// Mitsubishi GX Works2 project: DATN   PLC: FX3U/FX3UC

PROGRAM MAIN
VAR
  Retrieval_1 : Retrieval;
  Storage : Storage;
  Home_Sto_1 : Home_Sto;
  GoToFailPos_1 : GoToFailPos;
END_VAR
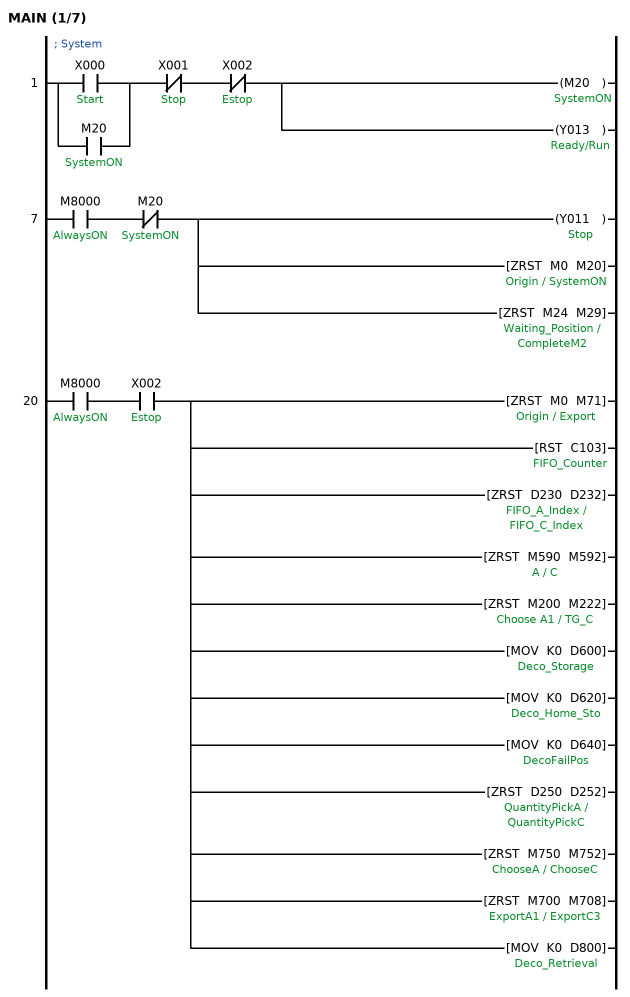
; System
1     LD      X000  ; Start
      OR      M20  ; SystemON
      ANI     X001  ; Stop
      ANI     X002  ; Estop
      OUT     M20  ; SystemON
      OUT     Y013  ; Ready/Run
7     LD      M8000  ; AlwaysON
      ANI     M20  ; SystemON
      OUT     Y011  ; Stop
      ZRST    M0 M20  ; Origin
      ZRST    M24 M29  ; Waiting_Position / CompleteM2
20    LD      M8000  ; AlwaysON
      AND     X002  ; Estop
      ZRST    M0 M71  ; Export
      RST     C103  ; FIFO_Counter
      ZRST    D230 D232  ; FIFO_A_Index / FIFO_C_Index
      ZRST    M590 M592  ; A / C
      ZRST    M200 M222  ; Choose A1 / TG_C
      MOV     K0 D600  ; Deco_Storage
      MOV     K0 D620  ; Deco_Home_Sto
      MOV     K0 D640  ; DecoFailPos
      ZRST    D250 D252  ; QuantityPickA / QuantityPickC
      ZRST    M750 M752  ; ChooseA / ChooseC
      ZRST    M700 M708  ; ExportA1 / ExportC3
      MOV     K0 D800  ; Deco_Retrieval
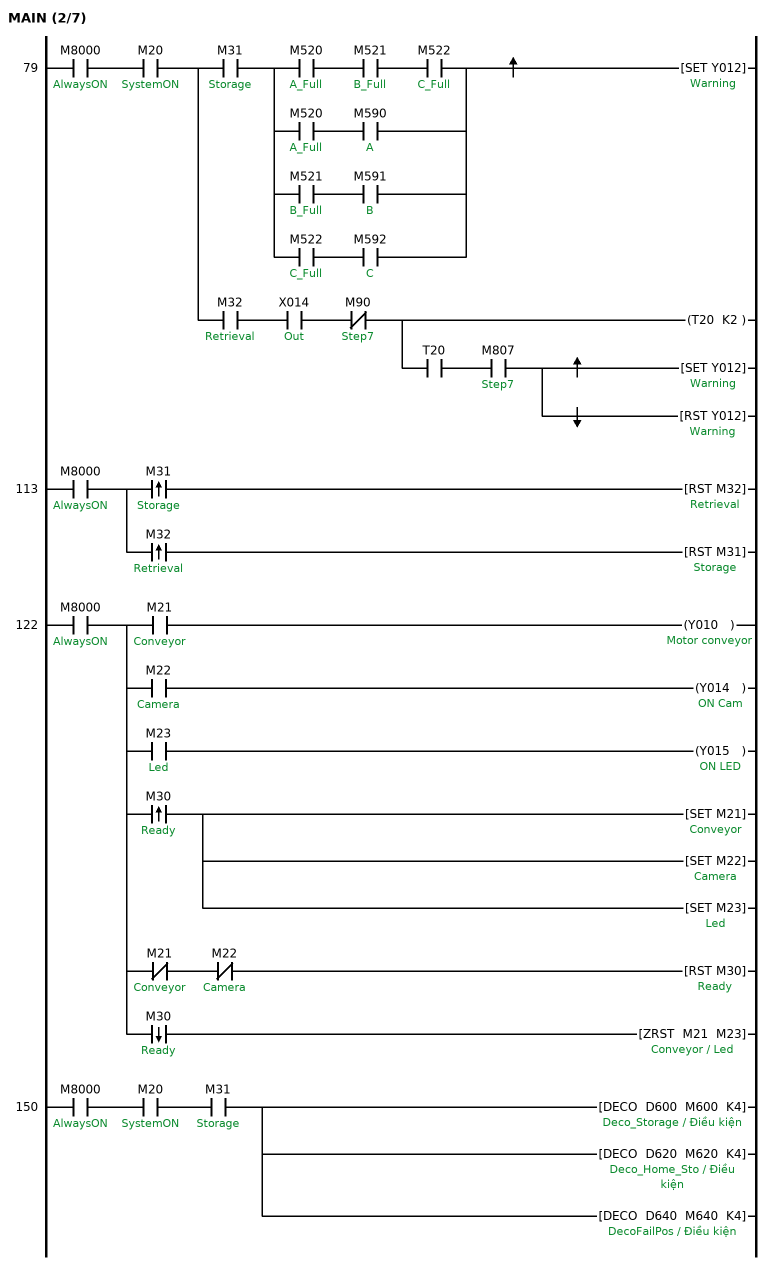
79    LD      M8000  ; AlwaysON
      AND     M20  ; SystemON
      MPS
      AND     M31  ; Storage
      LD      M520  ; A_Full
      AND     M521  ; B_Full
      AND     M522  ; C_Full
      LD      M520  ; A_Full
      AND     M590  ; A
      ORB
      LD      M521  ; B_Full
      AND     M591  ; B
      ORB
      LD      M522  ; C_Full
      AND     M592  ; C
      ORB
      ANB
      MEP
      SET     Y012  ; Warning
      MPP
      AND     M32  ; Retrieval
      AND     X014  ; Out
      ANI     M90  ; Step7
      OUT     T20 K2
      AND     T20
      AND     M807  ; Step7
      MPS
      MEP
      SET     Y012  ; Warning
      MPP
      MEF
      RST     Y012  ; Warning
113   LD      M8000  ; AlwaysON
      MPS
      ANDP    M31  ; Storage
      RST     M32  ; Retrieval
      MPP
      ANDP    M32  ; Retrieval
      RST     M31  ; Storage
122   LD      M8000  ; AlwaysON
      MPS
      AND     M21  ; Conveyor
      OUT     Y010  ; Motor conveyor
      MRD
      AND     M22  ; Camera
      OUT     Y014  ; ON Cam
      MRD
      AND     M23  ; Led
      OUT     Y015  ; ON LED
      MRD
      ANDP    M30  ; Ready
      SET     M21  ; Conveyor
      SET     M22  ; Camera
      SET     M23  ; Led
      MRD
      ANI     M21  ; Conveyor
      ANI     M22  ; Camera
      RST     M30  ; Ready
      MPP
      ANDF    M30  ; Ready
      ZRST    M21 M23
150   LD      M8000  ; AlwaysON
      AND     M20  ; SystemON
      AND     M31  ; Storage
      DECO    D600 M600 K4  ; Điều kiện
      DECO    D620 M620 K4  ; Điều kiện
      DECO    D640 M640 K4  ; Điều kiện
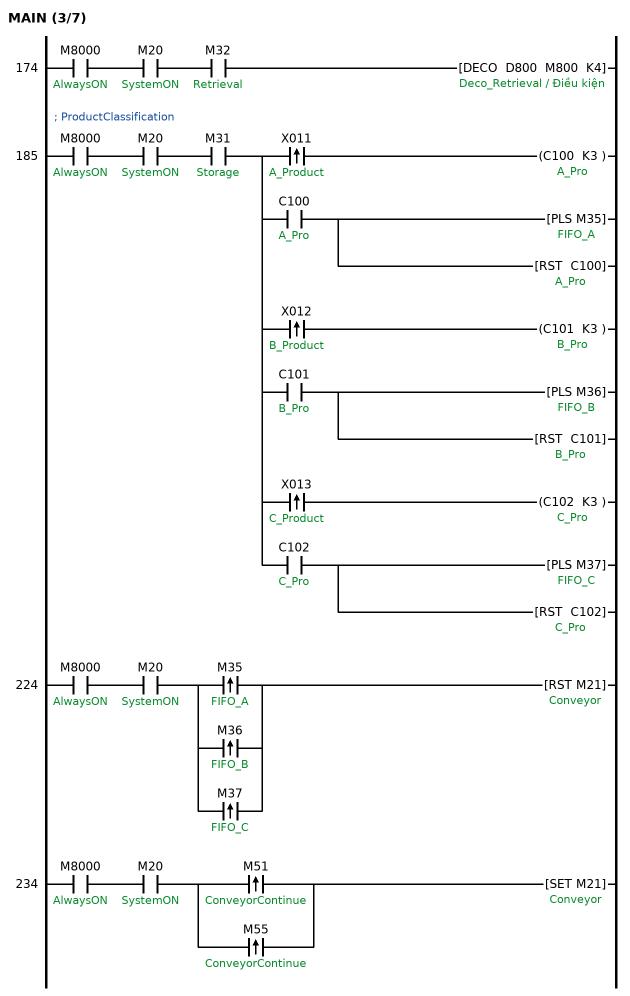
174   LD      M8000  ; AlwaysON
      AND     M20  ; SystemON
      AND     M32  ; Retrieval
      DECO    D800 M800 K4  ; Điều kiện
; ProductClassification
185   LD      M8000  ; AlwaysON
      AND     M20  ; SystemON
      AND     M31  ; Storage
      MPS
      ANDP    X011  ; A_Product
      OUT     C100 K3  ; A_Pro
      MRD
      AND     C100  ; A_Pro
      PLS     M35  ; FIFO_A
      RST     C100  ; A_Pro
      MRD
      ANDP    X012  ; B_Product
      OUT     C101 K3  ; B_Pro
      MRD
      AND     C101  ; B_Pro
      PLS     M36  ; FIFO_B
      RST     C101  ; B_Pro
      MRD
      ANDP    X013  ; C_Product
      OUT     C102 K3  ; C_Pro
      MPP
      AND     C102  ; C_Pro
      PLS     M37  ; FIFO_C
      RST     C102  ; C_Pro
224   LD      M8000  ; AlwaysON
      AND     M20  ; SystemON
      LDP     M35  ; FIFO_A
      ORP     M36  ; FIFO_B
      ORP     M37  ; FIFO_C
      ANB
      RST     M21  ; Conveyor
234   LD      M8000  ; AlwaysON
      AND     M20  ; SystemON
      LDP     M51  ; ConveyorContinue
      ORP     M55  ; ConveyorContinue
      ANB
      SET     M21  ; Conveyor
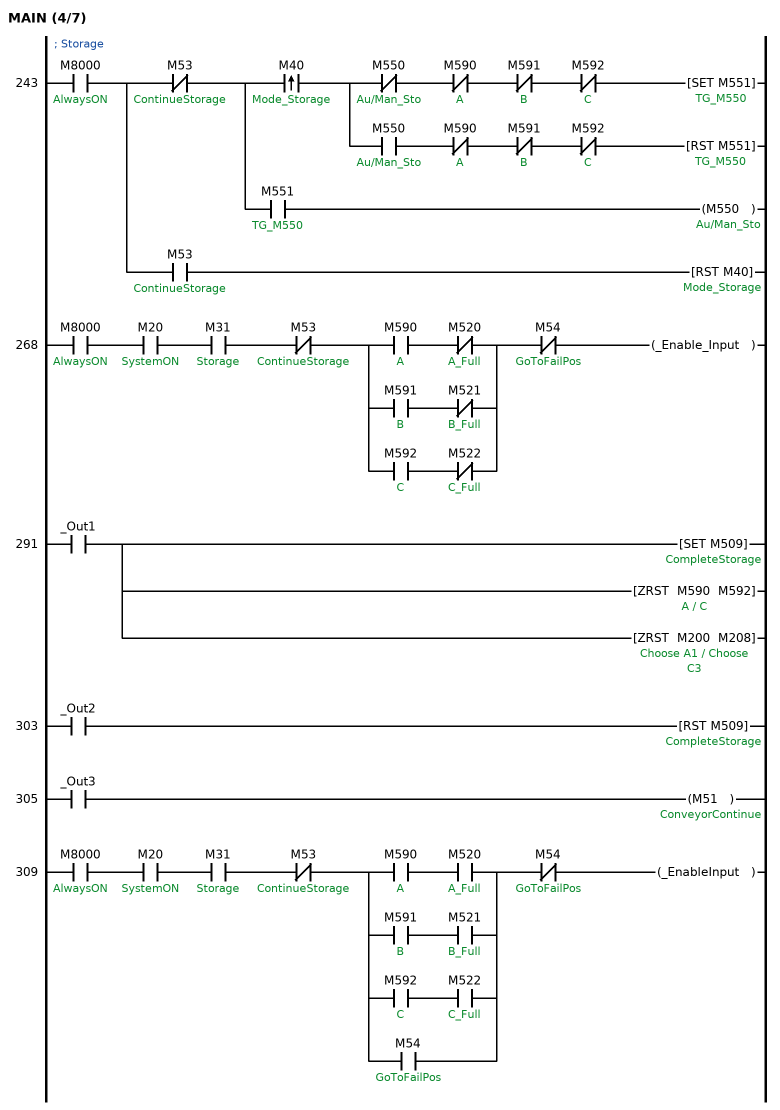
; Storage
243   LD      M8000  ; AlwaysON
      MPS
      ANI     M53  ; ContinueStorage
      MPS
      ANDP    M40  ; Mode_Storage
      MPS
      ANI     M550  ; Au/Man_Sto
      ANI     M590  ; A
      ANI     M591  ; B
      ANI     M592  ; C
      SET     M551  ; TG_M550
      MPP
      AND     M550  ; Au/Man_Sto
      ANI     M590  ; A
      ANI     M591  ; B
      ANI     M592  ; C
      RST     M551  ; TG_M550
      MPP
      AND     M551  ; TG_M550
      OUT     M550  ; Au/Man_Sto
      MPP
      AND     M53  ; ContinueStorage
      RST     M40  ; Mode_Storage
; FB BLK START Storage(Storage)
268   LD      M8000  ; AlwaysON
      AND     M20  ; SystemON
      AND     M31  ; Storage
      ANI     M53  ; ContinueStorage
      LD      M590  ; A
      ANI     M520  ; A_Full
      LD      M591  ; B
      ANI     M521  ; B_Full
      ORB
      LD      M592  ; C
      ANI     M522  ; C_Full
      ORB
      ANB
      ANI     M54  ; GoToFailPos
      OUT     _Enable_Input
; FB START
; FB_NAME Storage
; INSTANCE_NAME Storage
; FB IN_B:Enable_Input
; FB OUT_Out1:B
; FB OUT_Out2:B
; FB OUT_Out3:B
; FB END
291   LD      _Out1
      SET     M509  ; CompleteStorage
      ZRST    M590 M592
      ZRST    M200 M208  ; Choose C3
303   LD      _Out2
      RST     M509  ; CompleteStorage
305   LD      _Out3
      OUT     M51  ; ConveyorContinue
; FB BLK END
; FB BLK START Home_Sto(Home_Sto_1)
309   LD      M8000  ; AlwaysON
      AND     M20  ; SystemON
      AND     M31  ; Storage
      ANI     M53  ; ContinueStorage
      LD      M590  ; A
      AND     M520  ; A_Full
      LD      M591  ; B
      AND     M521  ; B_Full
      ORB
      LD      M592  ; C
      AND     M522  ; C_Full
      ORB
      OR      M54  ; GoToFailPos
      ANB
      ANI     M54  ; GoToFailPos
      OUT     _EnableInput
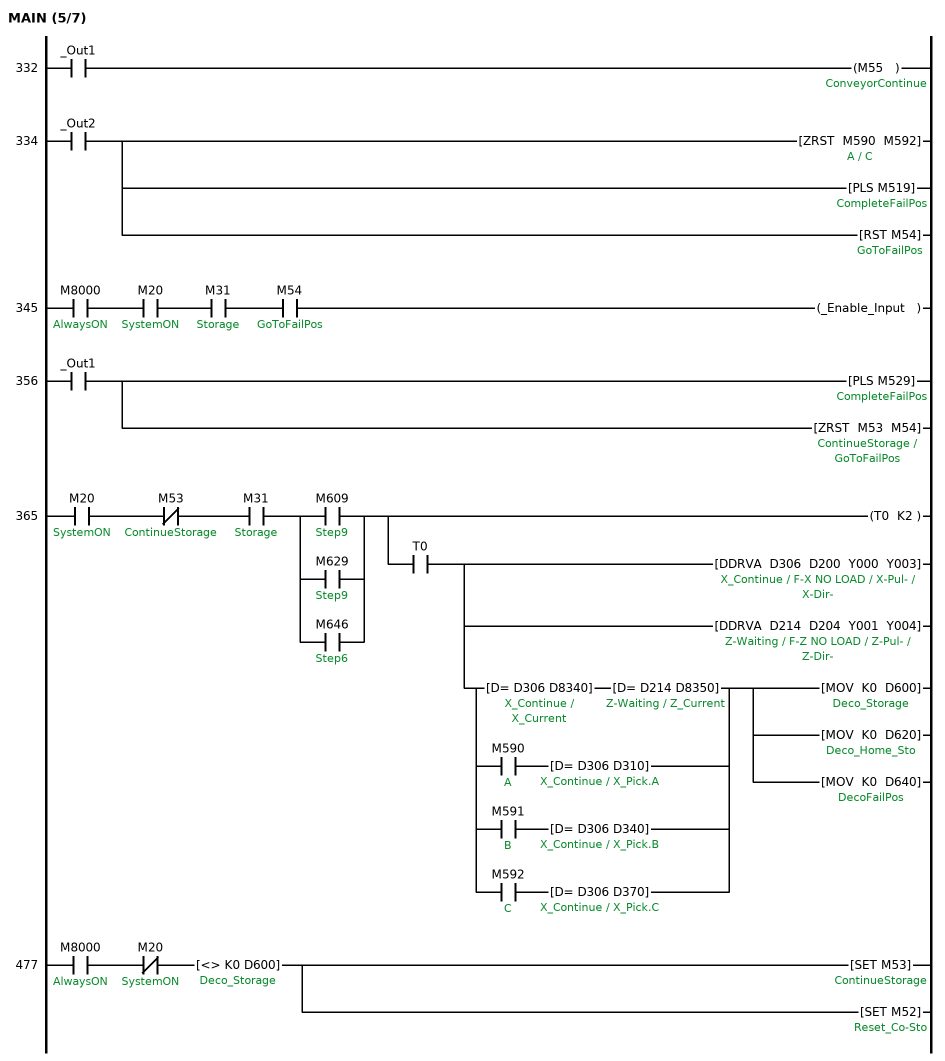
; FB START
; FB_NAME Home_Sto
; INSTANCE_NAME Home_Sto_1
; FB IN_B:EnableInput
; FB OUT_Out1:B
; FB OUT_Out2:B
; FB END
332   LD      _Out1
      OUT     M55  ; ConveyorContinue
334   LD      _Out2
      ZRST    M590 M592
      PLS     M519  ; CompleteFailPos
      RST     M54  ; GoToFailPos
; FB BLK END
; FB BLK START GoToFailPos(GoToFailPos_1)
345   LD      M8000  ; AlwaysON
      AND     M20  ; SystemON
      AND     M31  ; Storage
      AND     M54  ; GoToFailPos
      OUT     _Enable_Input
; FB START
; FB_NAME GoToFailPos
; INSTANCE_NAME GoToFailPos_1
; FB IN_B:Enable_Input
; FB OUT_Out1:B
; FB END
356   LD      _Out1
      PLS     M529  ; CompleteFailPos
      ZRST    M53 M54
; FB BLK END
365   LD      M20  ; SystemON
      ANI     M53  ; ContinueStorage
      AND     M31  ; Storage
      LD      M609  ; Step9
      OR      M629  ; Step9
      OR      M646  ; Step6
      ANB
      OUT     T0 K2
      AND     T0
      DDRVA   D306 D200 Y000 Y003  ; X_Continue / F-X NO LOAD / X-Pul- / X-Dir-
      DDRVA   D214 D204 Y001 Y004  ; Z-Waiting / F-Z NO LOAD / Z-Pul- / Z-Dir-
      LDD=    D306 D8340  ; X_Continue / X_Current
      ANDD=   D214 D8350  ; Z-Waiting / Z_Current
      LD      M590  ; A
      ANDD=   D306 D310  ; X_Continue / X_Pick.A
      ORB
      LD      M591  ; B
      ANDD=   D306 D340  ; X_Continue / X_Pick.B
      ORB
      LD      M592  ; C
      ANDD=   D306 D370  ; X_Continue / X_Pick.C
      ORB
      ANB
      MOV     K0 D600
      MOV     K0 D620
      MOV     K0 D640
477   LD      M8000  ; AlwaysON
      ANI     M20  ; SystemON
      AND<>   K0 D600  ; Deco_Storage
      SET     M53  ; ContinueStorage
      SET     M52  ; Reset_Co-Sto
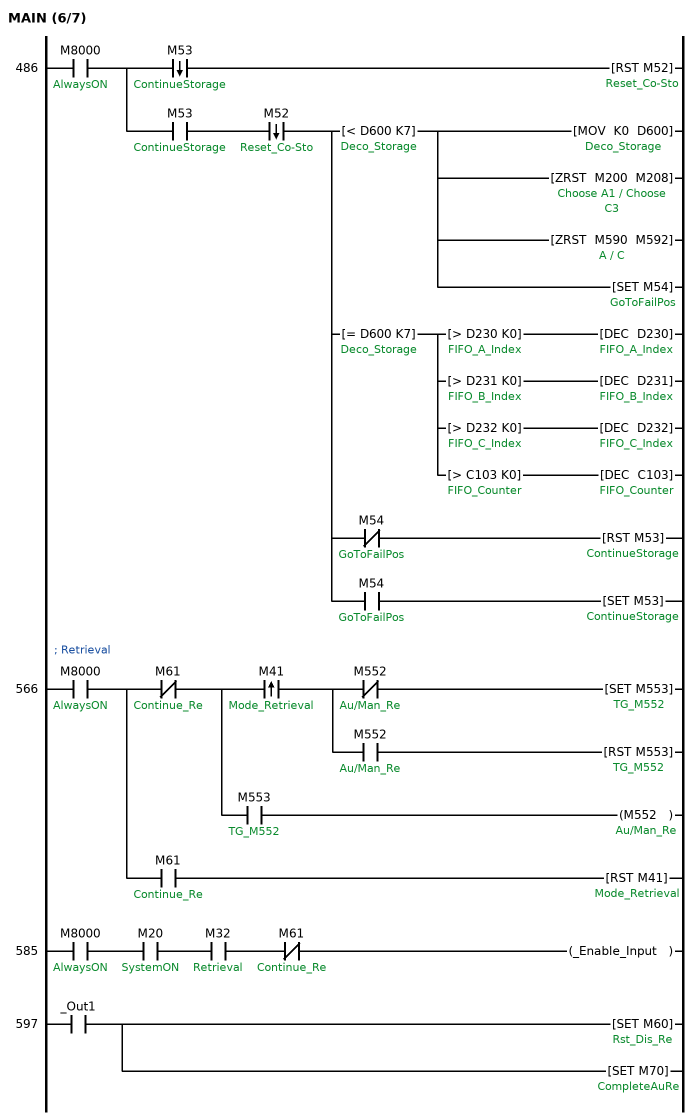
486   LD      M8000  ; AlwaysON
      MPS
      ANDF    M53  ; ContinueStorage
      RST     M52  ; Reset_Co-Sto
      MPP
      AND     M53  ; ContinueStorage
      ANDF    M52  ; Reset_Co-Sto
      MPS
      AND<    D600 K7  ; Deco_Storage
      MOV     K0 D600
      ZRST    M200 M208
      ZRST    M590 M592
      SET     M54  ; GoToFailPos
      MRD
      AND=    D600 K7  ; Deco_Storage
      MPS
      AND>    D230 K0  ; FIFO_A_Index
      DEC     D230
      MRD
      AND>    D231 K0  ; FIFO_B_Index
      DEC     D231
      MRD
      AND>    D232 K0  ; FIFO_C_Index
      DEC     D232
      MPP
      AND>    C103 K0  ; FIFO_Counter
      DEC     C103
      MRD
      ANI     M54  ; GoToFailPos
      RST     M53  ; ContinueStorage
      MPP
      AND     M54  ; GoToFailPos
      SET     M53  ; ContinueStorage
; Retrieval
566   LD      M8000  ; AlwaysON
      MPS
      ANI     M61  ; Continue_Re
      MPS
      ANDP    M41  ; Mode_Retrieval
      MPS
      ANI     M552  ; Au/Man_Re
      SET     M553  ; TG_M552
      MPP
      AND     M552  ; Au/Man_Re
      RST     M553  ; TG_M552
      MPP
      AND     M553  ; TG_M552
      OUT     M552  ; Au/Man_Re
      MPP
      AND     M61  ; Continue_Re
      RST     M41  ; Mode_Retrieval
; FB BLK START Retrieval(Retrieval_1)
585   LD      M8000  ; AlwaysON
      AND     M20  ; SystemON
      AND     M32  ; Retrieval
      ANI     M61  ; Continue_Re
      OUT     _Enable_Input
; FB START
; FB_NAME Retrieval
; INSTANCE_NAME Retrieval_1
; FB IN_B:Enable_Input
; FB OUT_Out1:B
; FB OUT_Out2:B
; FB END
597   LD      _Out1
      SET     M60  ; Rst_Dis_Re
      SET     M70  ; CompleteAuRe
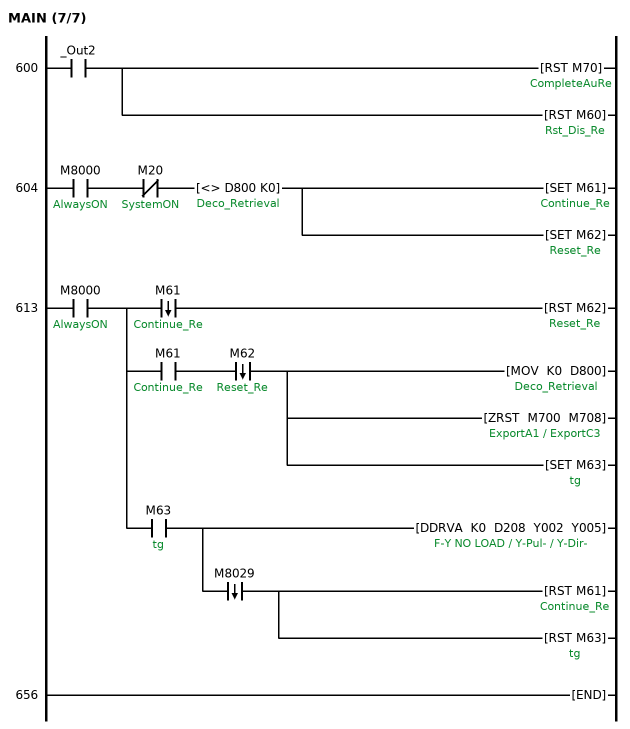
600   LD      _Out2
      RST     M70  ; CompleteAuRe
      RST     M60  ; Rst_Dis_Re
; FB BLK END
604   LD      M8000  ; AlwaysON
      ANI     M20  ; SystemON
      AND<>   D800 K0  ; Deco_Retrieval
      SET     M61  ; Continue_Re
      SET     M62  ; Reset_Re
613   LD      M8000  ; AlwaysON
      MPS
      ANDF    M61  ; Continue_Re
      RST     M62  ; Reset_Re
      MRD
      AND     M61  ; Continue_Re
      ANDF    M62  ; Reset_Re
      MOV     K0 D800
      ZRST    M700 M708
      SET     M63  ; tg
      MPP
      AND     M63  ; tg
      DDRVA   K0 D208 Y002 Y005  ; F-Y NO LOAD / Y-Pul- / Y-Dir-
      ANDF    M8029
      RST     M61  ; Continue_Re
      RST     M63  ; tg
656   END
END_PROGRAM

PROGRAM HOME
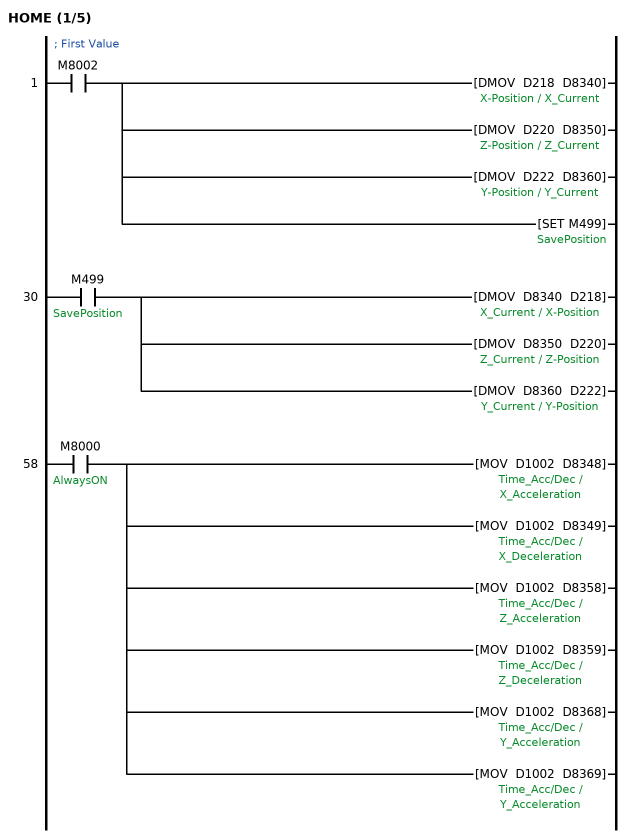
; First Value
1     LD      M8002
      DMOV    D218 D8340  ; X-Position / X_Current
      DMOV    D220 D8350  ; Z-Position / Z_Current
      DMOV    D222 D8360  ; Y-Position / Y_Current
      SET     M499  ; SavePosition
30    LD      M499  ; SavePosition
      DMOV    D8340 D218
      DMOV    D8350 D220
      DMOV    D8360 D222
58    LD      M8000  ; AlwaysON
      MOV     D1002 D8348  ; Time_Acc/Dec / X_Acceleration
      MOV     D1002 D8349  ; X_Deceleration
      MOV     D1002 D8358  ; Z_Acceleration
      MOV     D1002 D8359  ; Z_Deceleration
      MOV     D1002 D8368  ; Y_Acceleration
      MOV     D1002 D8369  ; Y_Acceleration
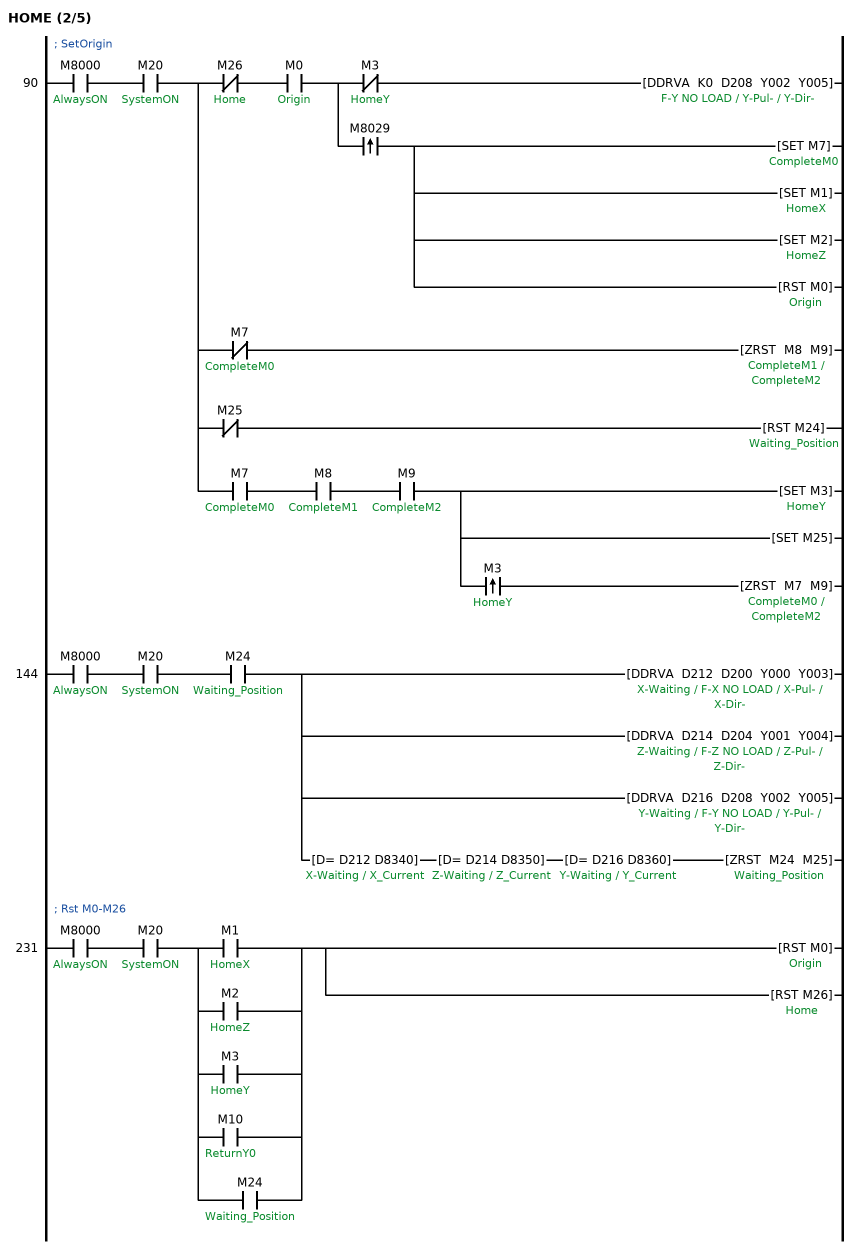
; SetOrigin
90    LD      M8000  ; AlwaysON
      AND     M20  ; SystemON
      MPS
      ANI     M26  ; Home
      AND     M0  ; Origin
      MPS
      ANI     M3  ; HomeY
      DDRVA   K0 D208 Y002 Y005  ; F-Y NO LOAD / Y-Pul- / Y-Dir-
      MPP
      ANDP    M8029
      SET     M7  ; CompleteM0
      SET     M1  ; HomeX
      SET     M2  ; HomeZ
      RST     M0  ; Origin
      MRD
      ANI     M7  ; CompleteM0
      ZRST    M8 M9  ; CompleteM1 / CompleteM2
      MRD
      ANI     M25
      RST     M24  ; Waiting_Position
      MPP
      AND     M7  ; CompleteM0
      AND     M8  ; CompleteM1
      AND     M9  ; CompleteM2
      SET     M3  ; HomeY
      SET     M25
      ANDP    M3  ; HomeY
      ZRST    M7 M9
144   LD      M8000  ; AlwaysON
      AND     M20  ; SystemON
      AND     M24  ; Waiting_Position
      DDRVA   D212 D200 Y000 Y003  ; X-Waiting / F-X NO LOAD / X-Pul- / X-Dir-
      DDRVA   D214 D204 Y001 Y004  ; Z-Waiting / F-Z NO LOAD / Z-Pul- / Z-Dir-
      DDRVA   D216 D208 Y002 Y005  ; Y-Waiting
      ANDD=   D212 D8340  ; X-Waiting / X_Current
      ANDD=   D214 D8350  ; Z-Waiting / Z_Current
      ANDD=   D216 D8360  ; Y-Waiting / Y_Current
      ZRST    M24 M25
; Rst M0-M26
231   LD      M8000  ; AlwaysON
      AND     M20  ; SystemON
      LD      M1  ; HomeX
      OR      M2  ; HomeZ
      OR      M3  ; HomeY
      OR      M10  ; ReturnY0
      OR      M24  ; Waiting_Position
      ANB
      RST     M0  ; Origin
      RST     M26  ; Home
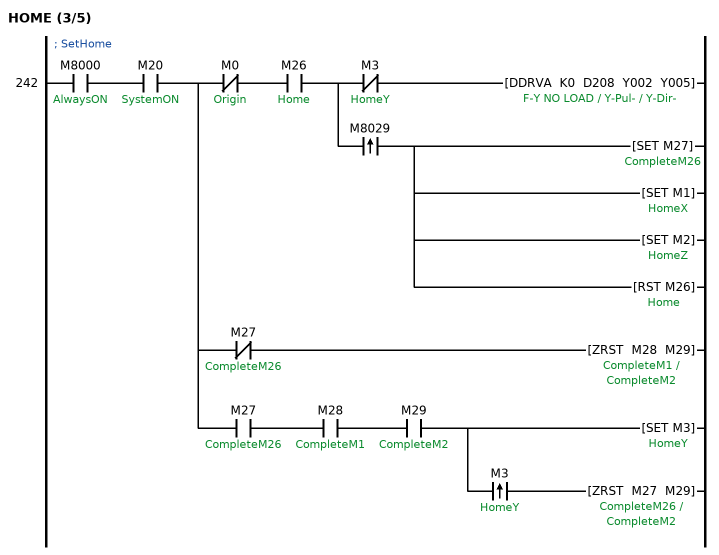
; SetHome
242   LD      M8000  ; AlwaysON
      AND     M20  ; SystemON
      MPS
      ANI     M0  ; Origin
      AND     M26  ; Home
      MPS
      ANI     M3  ; HomeY
      DDRVA   K0 D208 Y002 Y005
      MPP
      ANDP    M8029
      SET     M27  ; CompleteM26
      SET     M1  ; HomeX
      SET     M2  ; HomeZ
      RST     M26  ; Home
      MRD
      ANI     M27  ; CompleteM26
      ZRST    M28 M29  ; CompleteM1 / CompleteM2
      MPP
      AND     M27  ; CompleteM26
      AND     M28  ; CompleteM1
      AND     M29  ; CompleteM2
      SET     M3  ; HomeY
      ANDP    M3  ; HomeY
      ZRST    M27 M29
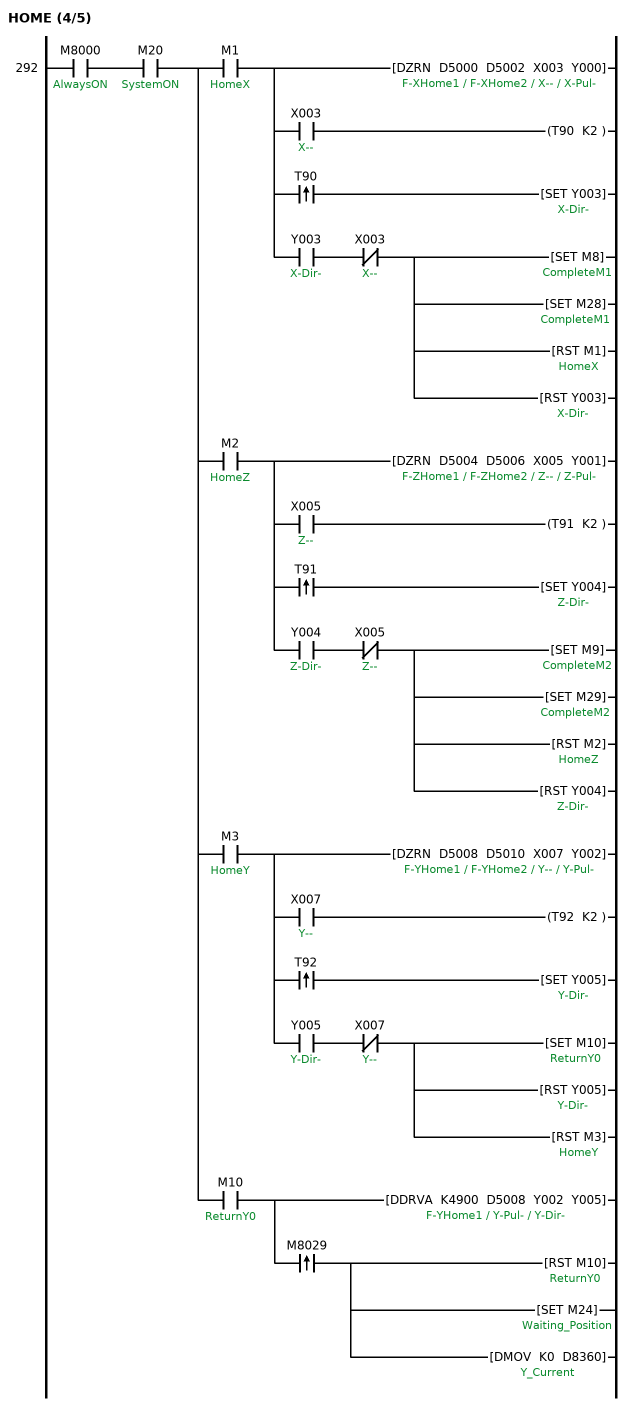
292   LD      M8000  ; AlwaysON
      AND     M20  ; SystemON
      MPS
      AND     M1  ; HomeX
      DZRN    D5000 D5002 X003 Y000  ; F-XHome1 / F-XHome2 / X--
      MPS
      AND     X003  ; X--
      OUT     T90 K2
      MRD
      ANDP    T90
      SET     Y003  ; X-Dir-
      MPP
      AND     Y003  ; X-Dir-
      ANI     X003  ; X--
      SET     M8  ; CompleteM1
      SET     M28  ; CompleteM1
      RST     M1  ; HomeX
      RST     Y003  ; X-Dir-
      MRD
      AND     M2  ; HomeZ
      DZRN    D5004 D5006 X005 Y001  ; F-ZHome1 / F-ZHome2 / Z--
      MPS
      AND     X005  ; Z--
      OUT     T91 K2
      MRD
      ANDP    T91
      SET     Y004  ; Z-Dir-
      MPP
      AND     Y004  ; Z-Dir-
      ANI     X005  ; Z--
      SET     M9  ; CompleteM2
      SET     M29  ; CompleteM2
      RST     M2  ; HomeZ
      RST     Y004  ; Z-Dir-
      MRD
      AND     M3  ; HomeY
      DZRN    D5008 D5010 X007 Y002  ; F-YHome1 / F-YHome2 / Y--
      MPS
      AND     X007  ; Y--
      OUT     T92 K2
      MRD
      ANDP    T92
      SET     Y005  ; Y-Dir-
      MPP
      AND     Y005  ; Y-Dir-
      ANI     X007  ; Y--
      SET     M10  ; ReturnY0
      RST     Y005  ; Y-Dir-
      RST     M3  ; HomeY
      MPP
      AND     M10  ; ReturnY0
      DDRVA   K4900 D5008 Y002 Y005
      ANDP    M8029
      RST     M10  ; ReturnY0
      SET     M24  ; Waiting_Position
      DMOV    K0 D8360
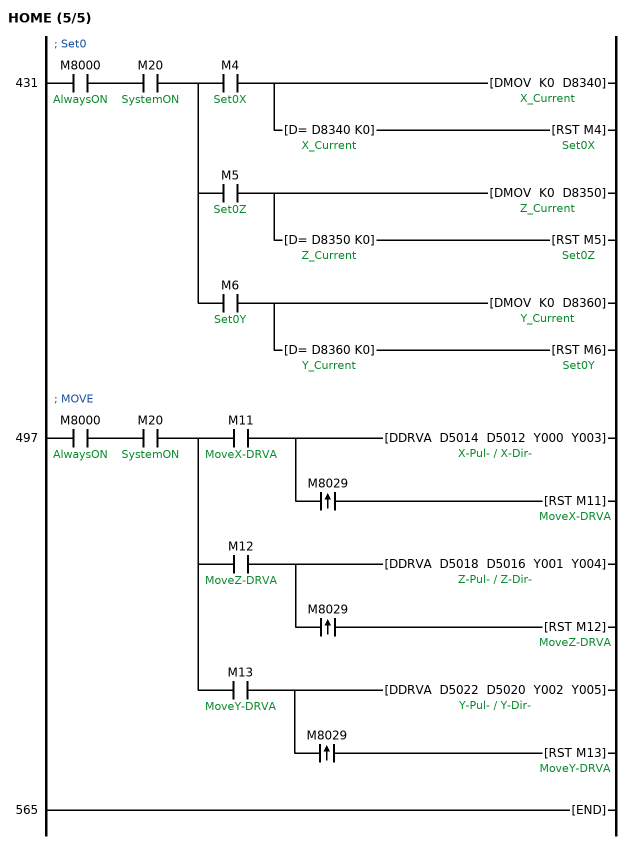
; Set0
431   LD      M8000  ; AlwaysON
      AND     M20  ; SystemON
      MPS
      AND     M4  ; Set0X
      DMOV    K0 D8340
      ANDD=   D8340 K0  ; X_Current
      RST     M4  ; Set0X
      MRD
      AND     M5  ; Set0Z
      DMOV    K0 D8350
      ANDD=   D8350 K0  ; Z_Current
      RST     M5  ; Set0Z
      MPP
      AND     M6  ; Set0Y
      DMOV    K0 D8360
      ANDD=   D8360 K0  ; Y_Current
      RST     M6  ; Set0Y
; MOVE
497   LD      M8000  ; AlwaysON
      AND     M20  ; SystemON
      MPS
      AND     M11  ; MoveX-DRVA
      DDRVA   D5014 D5012 Y000 Y003
      ANDP    M8029
      RST     M11  ; MoveX-DRVA
      MRD
      AND     M12  ; MoveZ-DRVA
      DDRVA   D5018 D5016 Y001 Y004
      ANDP    M8029
      RST     M12  ; MoveZ-DRVA
      MPP
      AND     M13  ; MoveY-DRVA
      DDRVA   D5022 D5020 Y002 Y005
      ANDP    M8029
      RST     M13  ; MoveY-DRVA
565   END
END_PROGRAM

FUNCTION_BLOCK Storage
VAR_INPUT
  Enable_Input : BOOL;
END_VAR
VAR_OUTPUT
  Out1 : BOOL;  (* Box Position *)
  Out2 : BOOL;  (* Complete *)
  Out3 : BOOL;  (* Conveyor_Continue *)
END_VAR
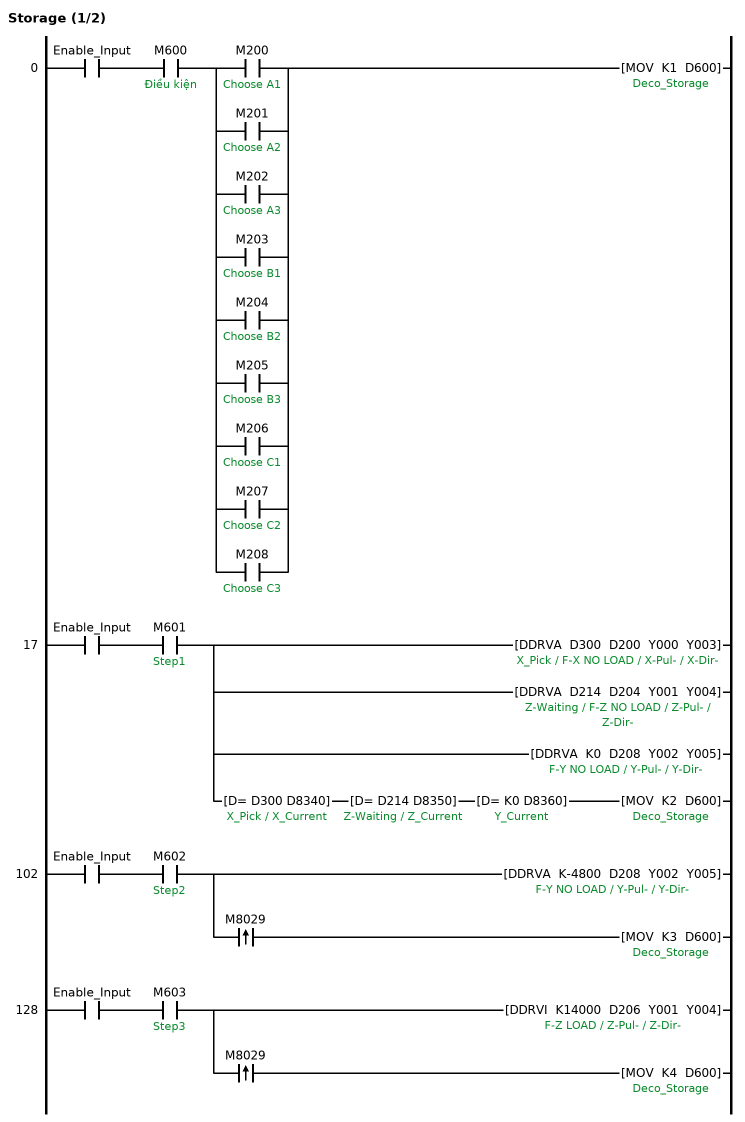
0     LD      Enable_Input
      AND     M600  ; Điều kiện
      LD      M200  ; Choose A1
      OR      M201  ; Choose A2
      OR      M202  ; Choose A3
      OR      M203  ; Choose B1
      OR      M204  ; Choose B2
      OR      M205  ; Choose B3
      OR      M206  ; Choose C1
      OR      M207  ; Choose C2
      OR      M208  ; Choose C3
      ANB
      MOV     K1 D600  ; Deco_Storage
17    LD      Enable_Input
      AND     M601  ; Step1
      DDRVA   D300 D200 Y000 Y003  ; X_Pick / F-X NO LOAD / X-Pul- / X-Dir-
      DDRVA   D214 D204 Y001 Y004  ; Z-Waiting / F-Z NO LOAD / Z-Pul- / Z-Dir-
      DDRVA   K0 D208 Y002 Y005  ; F-Y NO LOAD / Y-Pul- / Y-Dir-
      ANDD=   D300 D8340  ; X_Pick / X_Current
      ANDD=   D214 D8350  ; Z-Waiting / Z_Current
      ANDD=   K0 D8360  ; Y_Current
      MOV     K2 D600
102   LD      Enable_Input
      AND     M602  ; Step2
      DDRVA   K-4800 D208 Y002 Y005
      ANDP    M8029
      MOV     K3 D600
128   LD      Enable_Input
      AND     M603  ; Step3
      DDRVI   K14000 D206 Y001 Y004  ; F-Z LOAD
      ANDP    M8029
      MOV     K4 D600
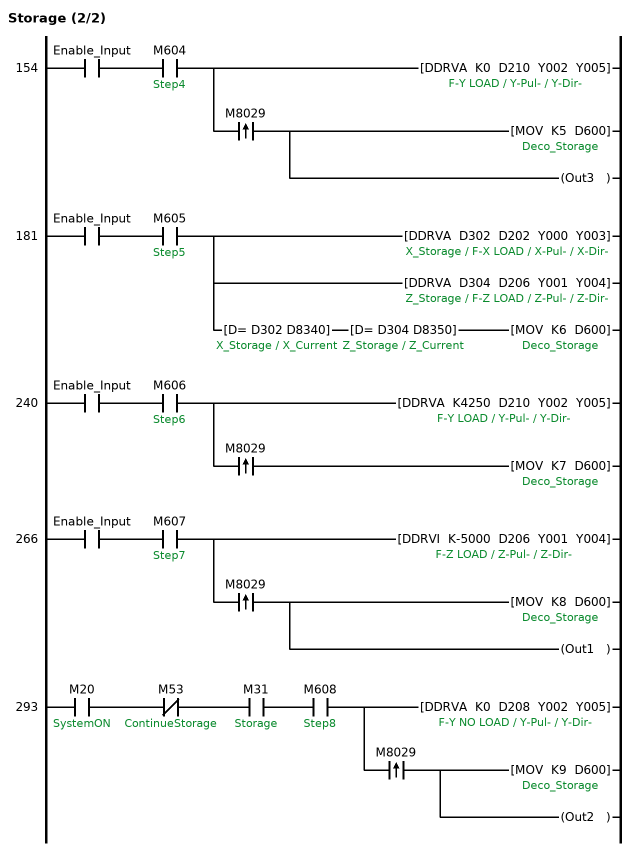
154   LD      Enable_Input
      AND     M604  ; Step4
      DDRVA   K0 D210 Y002 Y005  ; F-Y LOAD
      ANDP    M8029
      MOV     K5 D600
      OUT     Out3
181   LD      Enable_Input
      AND     M605  ; Step5
      DDRVA   D302 D202 Y000 Y003  ; X_Storage / F-X LOAD
      DDRVA   D304 D206 Y001 Y004  ; Z_Storage
      ANDD=   D302 D8340  ; X_Storage / X_Current
      ANDD=   D304 D8350  ; Z_Storage / Z_Current
      MOV     K6 D600
240   LD      Enable_Input
      AND     M606  ; Step6
      DDRVA   K4250 D210 Y002 Y005
      ANDP    M8029
      MOV     K7 D600
266   LD      Enable_Input
      AND     M607  ; Step7
      DDRVI   K-5000 D206 Y001 Y004
      ANDP    M8029
      MOV     K8 D600
      OUT     Out1
293   LD      M20  ; SystemON
      ANI     M53  ; ContinueStorage
      AND     M31  ; Storage
      AND     M608  ; Step8
      DDRVA   K0 D208 Y002 Y005
      ANDP    M8029
      MOV     K9 D600
      OUT     Out2
END_FUNCTION_BLOCK

PROGRAM Pos_Box
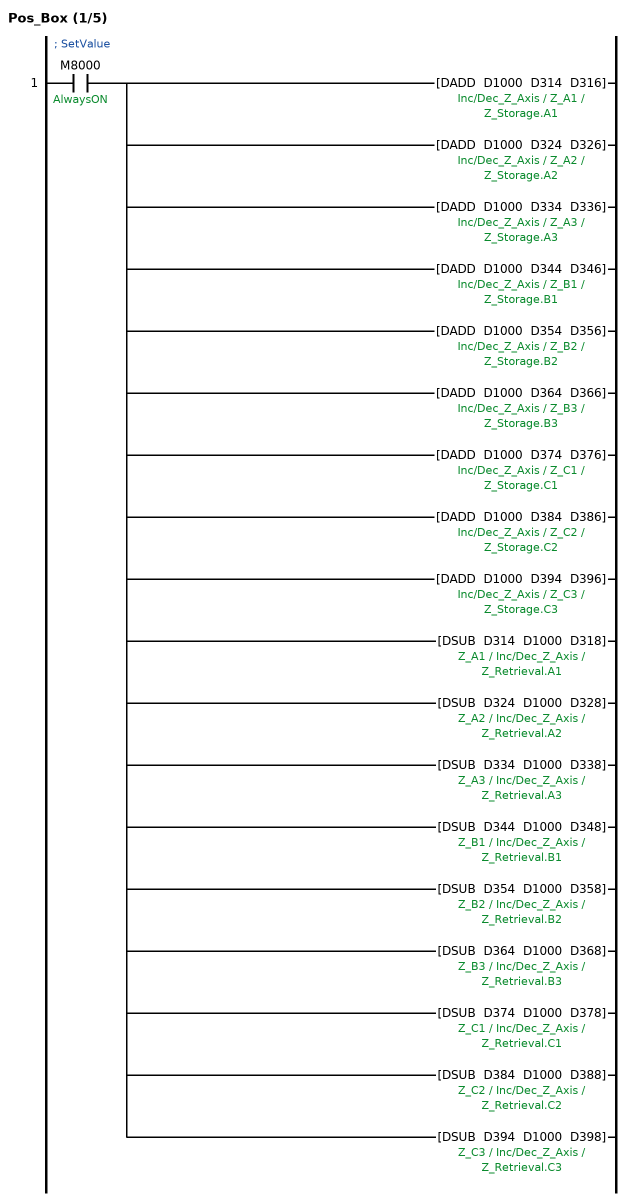
; SetValue
1     LD      M8000  ; AlwaysON
      DADD    D1000 D314 D316  ; Inc/Dec_Z_Axis / Z_A1 / Z_Storage.A1
      DADD    D1000 D324 D326  ; Z_A2 / Z_Storage.A2
      DADD    D1000 D334 D336  ; Z_A3 / Z_Storage.A3
      DADD    D1000 D344 D346  ; Z_B1 / Z_Storage.B1
      DADD    D1000 D354 D356  ; Z_B2 / Z_Storage.B2
      DADD    D1000 D364 D366  ; Z_B3 / Z_Storage.B3
      DADD    D1000 D374 D376  ; Z_C1 / Z_Storage.C1
      DADD    D1000 D384 D386  ; Z_C2 / Z_Storage.C2
      DADD    D1000 D394 D396  ; Z_C3 / Z_Storage.C3
      DSUB    D314 D1000 D318  ; Z_Retrieval.A1
      DSUB    D324 D1000 D328  ; Z_Retrieval.A2
      DSUB    D334 D1000 D338  ; Z_Retrieval.A3
      DSUB    D344 D1000 D348  ; Z_Retrieval.B1
      DSUB    D354 D1000 D358  ; Z_Retrieval.B2
      DSUB    D364 D1000 D368  ; Z_Retrieval.B3
      DSUB    D374 D1000 D378  ; Z_Retrieval.C1
      DSUB    D384 D1000 D388  ; Z_Retrieval.C2
      DSUB    D394 D1000 D398  ; Z_Retrieval.C3
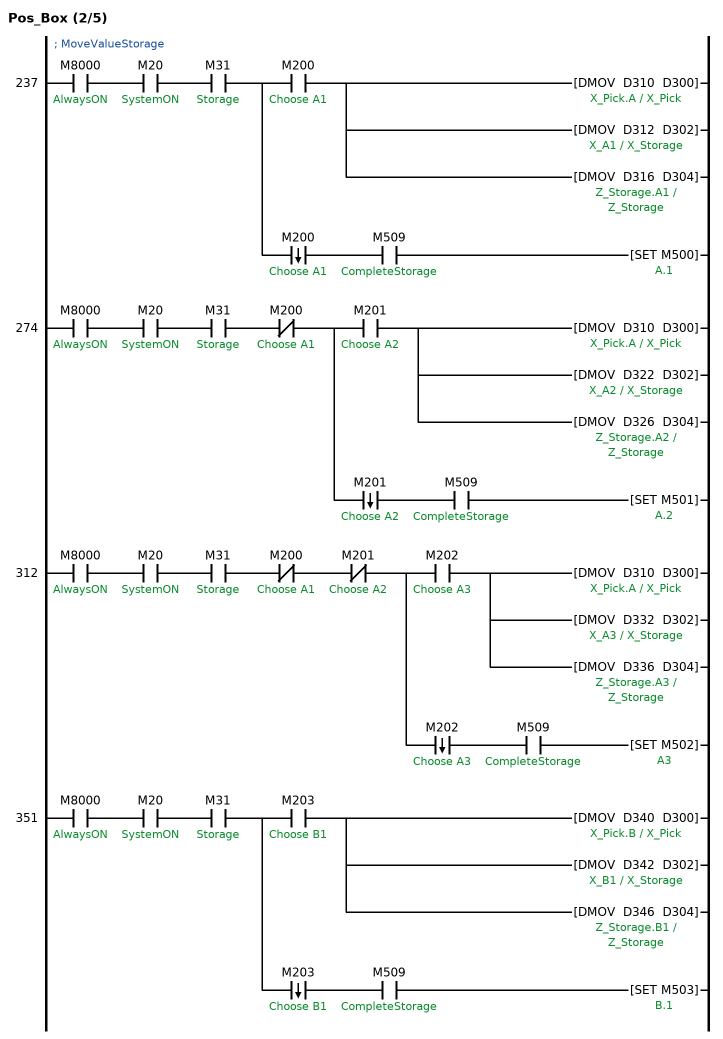
; MoveValueStorage
237   LD      M8000  ; AlwaysON
      AND     M20  ; SystemON
      AND     M31  ; Storage
      MPS
      AND     M200  ; Choose A1
      DMOV    D310 D300  ; X_Pick.A / X_Pick
      DMOV    D312 D302  ; X_A1 / X_Storage
      DMOV    D316 D304  ; Z_Storage
      MPP
      ANDF    M200  ; Choose A1
      AND     M509  ; CompleteStorage
      SET     M500  ; A.1
274   LD      M8000  ; AlwaysON
      AND     M20  ; SystemON
      AND     M31  ; Storage
      ANI     M200  ; Choose A1
      MPS
      AND     M201  ; Choose A2
      DMOV    D310 D300
      DMOV    D322 D302  ; X_A2
      DMOV    D326 D304
      MPP
      ANDF    M201  ; Choose A2
      AND     M509  ; CompleteStorage
      SET     M501  ; A.2
312   LD      M8000  ; AlwaysON
      AND     M20  ; SystemON
      AND     M31  ; Storage
      ANI     M200  ; Choose A1
      ANI     M201  ; Choose A2
      MPS
      AND     M202  ; Choose A3
      DMOV    D310 D300
      DMOV    D332 D302  ; X_A3
      DMOV    D336 D304
      MPP
      ANDF    M202  ; Choose A3
      AND     M509  ; CompleteStorage
      SET     M502  ; A3
351   LD      M8000  ; AlwaysON
      AND     M20  ; SystemON
      AND     M31  ; Storage
      MPS
      AND     M203  ; Choose B1
      DMOV    D340 D300  ; X_Pick.B
      DMOV    D342 D302  ; X_B1
      DMOV    D346 D304
      MPP
      ANDF    M203  ; Choose B1
      AND     M509  ; CompleteStorage
      SET     M503  ; B.1
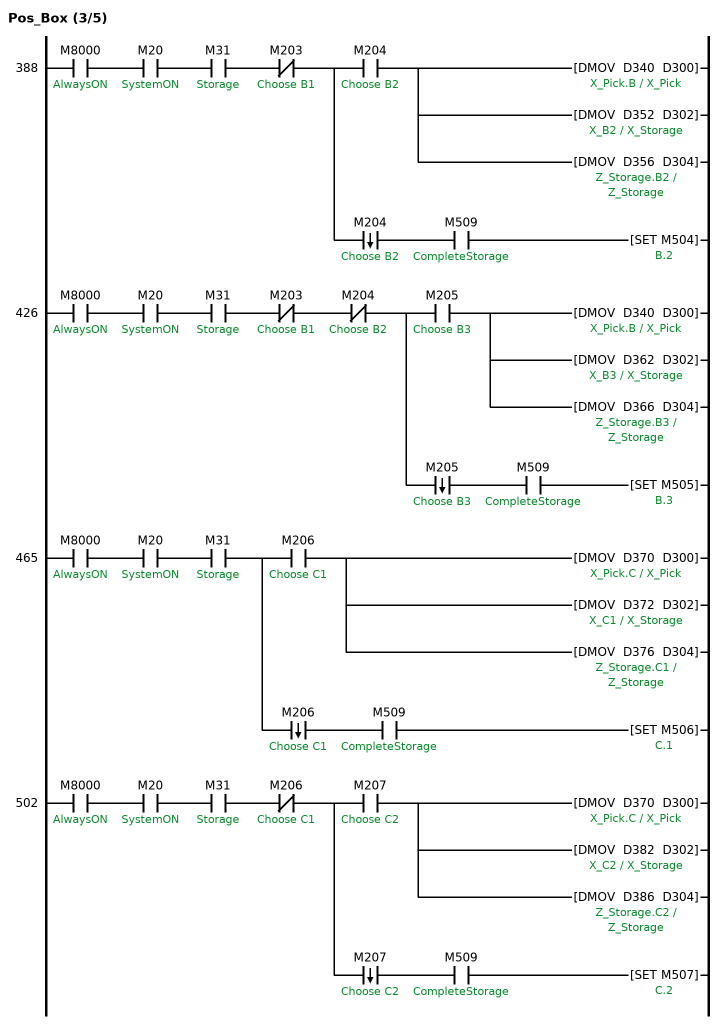
388   LD      M8000  ; AlwaysON
      AND     M20  ; SystemON
      AND     M31  ; Storage
      ANI     M203  ; Choose B1
      MPS
      AND     M204  ; Choose B2
      DMOV    D340 D300
      DMOV    D352 D302  ; X_B2
      DMOV    D356 D304
      MPP
      ANDF    M204  ; Choose B2
      AND     M509  ; CompleteStorage
      SET     M504  ; B.2
426   LD      M8000  ; AlwaysON
      AND     M20  ; SystemON
      AND     M31  ; Storage
      ANI     M203  ; Choose B1
      ANI     M204  ; Choose B2
      MPS
      AND     M205  ; Choose B3
      DMOV    D340 D300
      DMOV    D362 D302  ; X_B3
      DMOV    D366 D304
      MPP
      ANDF    M205  ; Choose B3
      AND     M509  ; CompleteStorage
      SET     M505  ; B.3
465   LD      M8000  ; AlwaysON
      AND     M20  ; SystemON
      AND     M31  ; Storage
      MPS
      AND     M206  ; Choose C1
      DMOV    D370 D300  ; X_Pick.C
      DMOV    D372 D302  ; X_C1
      DMOV    D376 D304
      MPP
      ANDF    M206  ; Choose C1
      AND     M509  ; CompleteStorage
      SET     M506  ; C.1
502   LD      M8000  ; AlwaysON
      AND     M20  ; SystemON
      AND     M31  ; Storage
      ANI     M206  ; Choose C1
      MPS
      AND     M207  ; Choose C2
      DMOV    D370 D300
      DMOV    D382 D302  ; X_C2
      DMOV    D386 D304
      MPP
      ANDF    M207  ; Choose C2
      AND     M509  ; CompleteStorage
      SET     M507  ; C.2
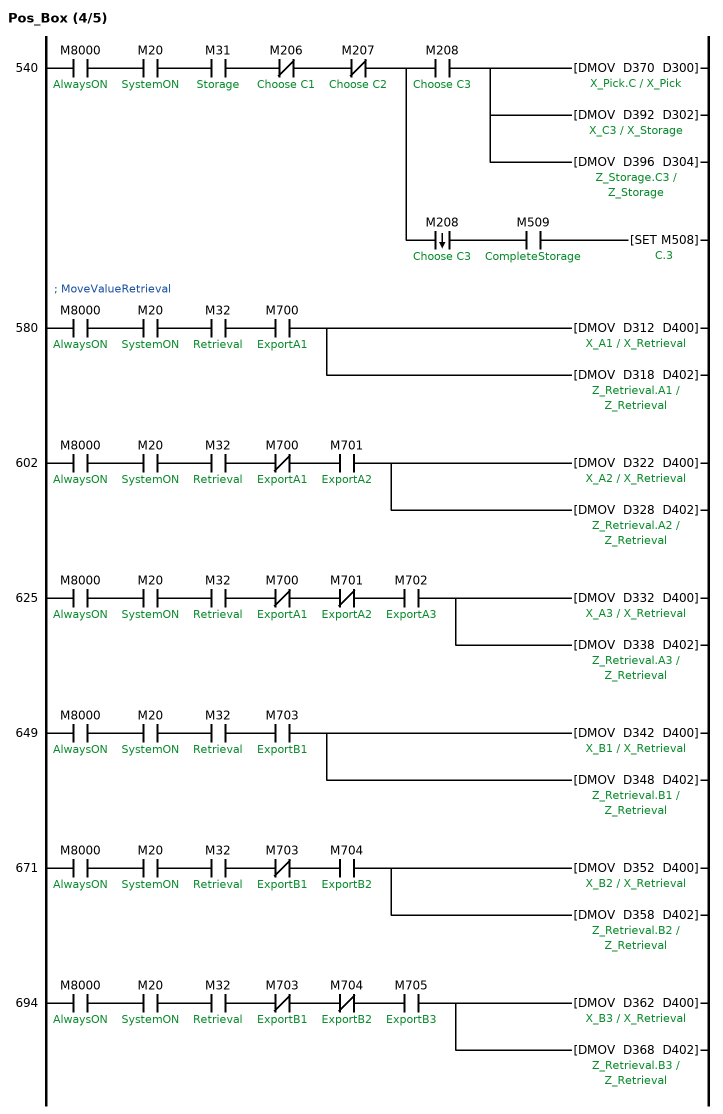
540   LD      M8000  ; AlwaysON
      AND     M20  ; SystemON
      AND     M31  ; Storage
      ANI     M206  ; Choose C1
      ANI     M207  ; Choose C2
      MPS
      AND     M208  ; Choose C3
      DMOV    D370 D300
      DMOV    D392 D302  ; X_C3
      DMOV    D396 D304
      MPP
      ANDF    M208  ; Choose C3
      AND     M509  ; CompleteStorage
      SET     M508  ; C.3
; MoveValueRetrieval
580   LD      M8000  ; AlwaysON
      AND     M20  ; SystemON
      AND     M32  ; Retrieval
      AND     M700  ; ExportA1
      DMOV    D312 D400  ; X_Retrieval
      DMOV    D318 D402  ; Z_Retrieval
602   LD      M8000  ; AlwaysON
      AND     M20  ; SystemON
      AND     M32  ; Retrieval
      ANI     M700  ; ExportA1
      AND     M701  ; ExportA2
      DMOV    D322 D400
      DMOV    D328 D402
625   LD      M8000  ; AlwaysON
      AND     M20  ; SystemON
      AND     M32  ; Retrieval
      ANI     M700  ; ExportA1
      ANI     M701  ; ExportA2
      AND     M702  ; ExportA3
      DMOV    D332 D400
      DMOV    D338 D402
649   LD      M8000  ; AlwaysON
      AND     M20  ; SystemON
      AND     M32  ; Retrieval
      AND     M703  ; ExportB1
      DMOV    D342 D400
      DMOV    D348 D402
671   LD      M8000  ; AlwaysON
      AND     M20  ; SystemON
      AND     M32  ; Retrieval
      ANI     M703  ; ExportB1
      AND     M704  ; ExportB2
      DMOV    D352 D400
      DMOV    D358 D402
694   LD      M8000  ; AlwaysON
      AND     M20  ; SystemON
      AND     M32  ; Retrieval
      ANI     M703  ; ExportB1
      ANI     M704  ; ExportB2
      AND     M705  ; ExportB3
      DMOV    D362 D400
      DMOV    D368 D402
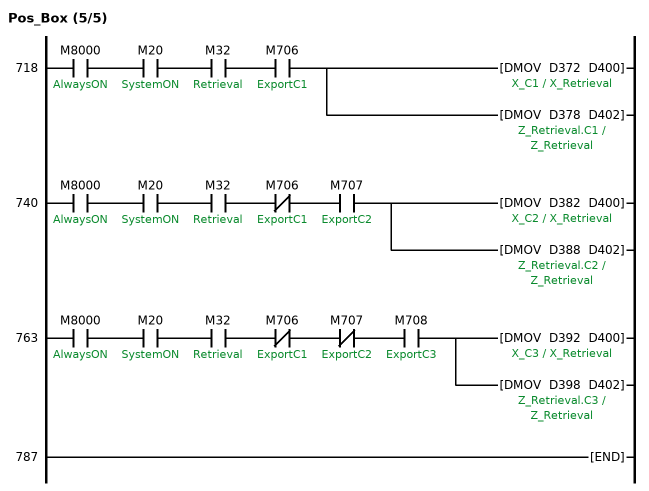
718   LD      M8000  ; AlwaysON
      AND     M20  ; SystemON
      AND     M32  ; Retrieval
      AND     M706  ; ExportC1
      DMOV    D372 D400
      DMOV    D378 D402
740   LD      M8000  ; AlwaysON
      AND     M20  ; SystemON
      AND     M32  ; Retrieval
      ANI     M706  ; ExportC1
      AND     M707  ; ExportC2
      DMOV    D382 D400
      DMOV    D388 D402
763   LD      M8000  ; AlwaysON
      AND     M20  ; SystemON
      AND     M32  ; Retrieval
      ANI     M706  ; ExportC1
      ANI     M707  ; ExportC2
      AND     M708  ; ExportC3
      DMOV    D392 D400
      DMOV    D398 D402
787   END
END_PROGRAM

FUNCTION_BLOCK Retrieval
VAR_INPUT
  Enable_Input : BOOL;
END_VAR
VAR_OUTPUT
  Out1 : BOOL;  (* RST_Display *)
  Out2 : BOOL;  (* RST *)
END_VAR
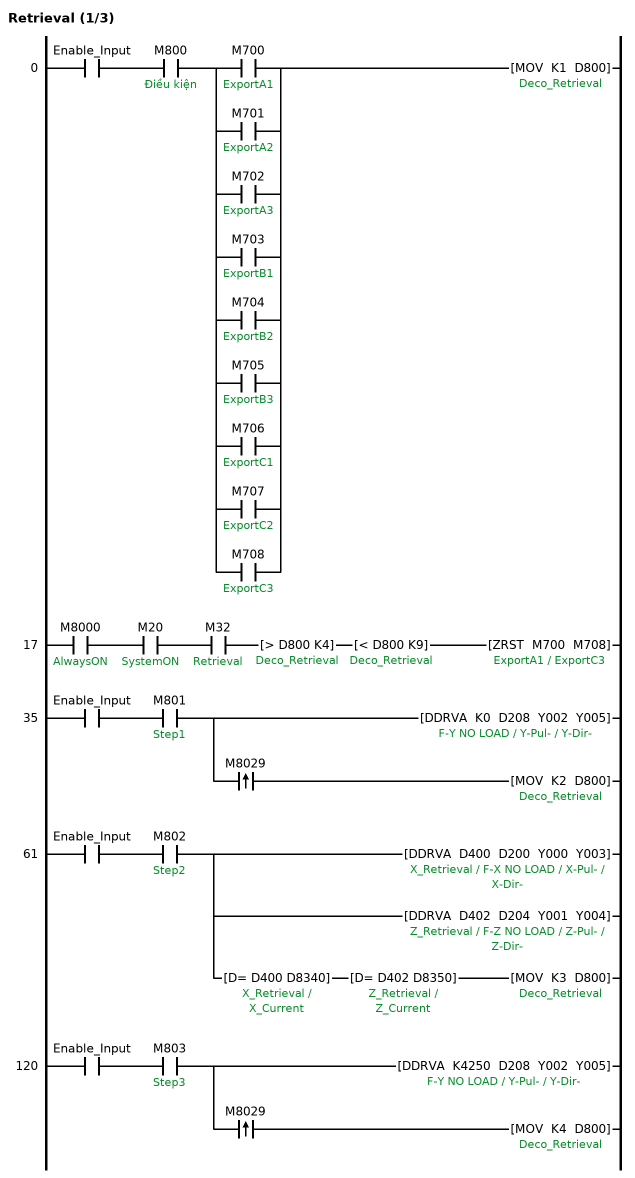
0     LD      Enable_Input
      AND     M800  ; Điều kiện
      LD      M700  ; ExportA1
      OR      M701  ; ExportA2
      OR      M702  ; ExportA3
      OR      M703  ; ExportB1
      OR      M704  ; ExportB2
      OR      M705  ; ExportB3
      OR      M706  ; ExportC1
      OR      M707  ; ExportC2
      OR      M708  ; ExportC3
      ANB
      MOV     K1 D800  ; Deco_Retrieval
17    LD      M8000  ; AlwaysON
      AND     M20  ; SystemON
      AND     M32  ; Retrieval
      AND>    D800 K4  ; Deco_Retrieval
      AND<    D800 K9  ; Deco_Retrieval
      ZRST    M700 M708
35    LD      Enable_Input
      AND     M801  ; Step1
      DDRVA   K0 D208 Y002 Y005  ; F-Y NO LOAD / Y-Pul- / Y-Dir-
      ANDP    M8029
      MOV     K2 D800
61    LD      Enable_Input
      AND     M802  ; Step2
      DDRVA   D400 D200 Y000 Y003  ; X_Retrieval / F-X NO LOAD / X-Pul- / X-Dir-
      DDRVA   D402 D204 Y001 Y004  ; Z_Retrieval / F-Z NO LOAD / Z-Pul- / Z-Dir-
      ANDD=   D400 D8340  ; X_Retrieval / X_Current
      ANDD=   D402 D8350  ; Z_Retrieval / Z_Current
      MOV     K3 D800
120   LD      Enable_Input
      AND     M803  ; Step3
      DDRVA   K4250 D208 Y002 Y005
      ANDP    M8029
      MOV     K4 D800
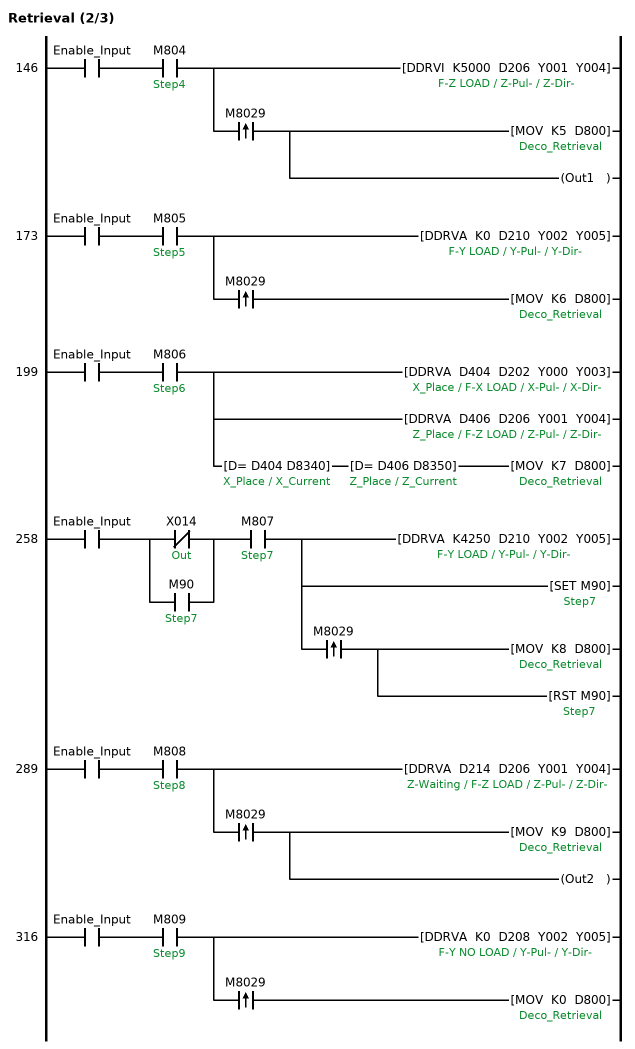
146   LD      Enable_Input
      AND     M804  ; Step4
      DDRVI   K5000 D206 Y001 Y004  ; F-Z LOAD
      ANDP    M8029
      MOV     K5 D800
      OUT     Out1
173   LD      Enable_Input
      AND     M805  ; Step5
      DDRVA   K0 D210 Y002 Y005  ; F-Y LOAD
      ANDP    M8029
      MOV     K6 D800
199   LD      Enable_Input
      AND     M806  ; Step6
      DDRVA   D404 D202 Y000 Y003  ; X_Place / F-X LOAD
      DDRVA   D406 D206 Y001 Y004  ; Z_Place
      ANDD=   D404 D8340  ; X_Place / X_Current
      ANDD=   D406 D8350  ; Z_Place / Z_Current
      MOV     K7 D800
258   LD      Enable_Input
      LDI     X014  ; Out
      OR      M90  ; Step7
      ANB
      AND     M807  ; Step7
      DDRVA   K4250 D210 Y002 Y005
      SET     M90  ; Step7
      ANDP    M8029
      MOV     K8 D800
      RST     M90  ; Step7
289   LD      Enable_Input
      AND     M808  ; Step8
      DDRVA   D214 D206 Y001 Y004  ; Z-Waiting
      ANDP    M8029
      MOV     K9 D800
      OUT     Out2
316   LD      Enable_Input
      AND     M809  ; Step9
      DDRVA   K0 D208 Y002 Y005
      ANDP    M8029
      MOV     K0 D800
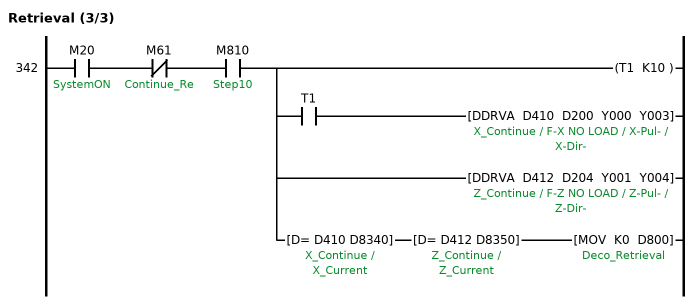
342   LD      M20  ; SystemON
      ANI     M61  ; Continue_Re
      AND     M810  ; Step10
      OUT     T1 K10
      MPS
      AND     T1
      DDRVA   D410 D200 Y000 Y003  ; X_Continue
      MPP
      DDRVA   D412 D204 Y001 Y004  ; Z_Continue
      ANDD=   D410 D8340  ; X_Continue / X_Current
      ANDD=   D412 D8350  ; Z_Continue / Z_Current
      MOV     K0 D800
END_FUNCTION_BLOCK

FUNCTION_BLOCK Home_Sto
VAR_INPUT
  EnableInput : BOOL;
END_VAR
VAR_OUTPUT
  Out2 : BOOL;  (* CompleteHomeSto *)
  Out1 : BOOL;  (* CompletePick *)
END_VAR
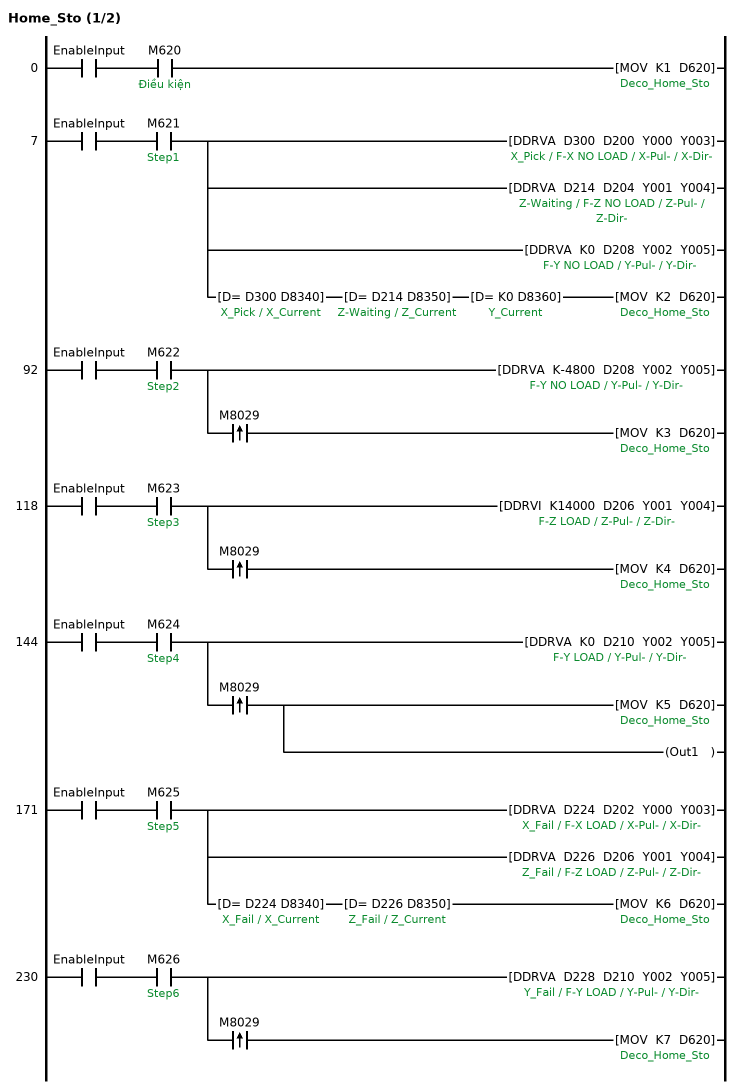
0     LD      EnableInput
      AND     M620  ; Điều kiện
      MOV     K1 D620  ; Deco_Home_Sto
7     LD      EnableInput
      AND     M621  ; Step1
      DDRVA   D300 D200 Y000 Y003  ; X_Pick / F-X NO LOAD / X-Pul- / X-Dir-
      DDRVA   D214 D204 Y001 Y004  ; Z-Waiting / F-Z NO LOAD / Z-Pul- / Z-Dir-
      DDRVA   K0 D208 Y002 Y005  ; F-Y NO LOAD / Y-Pul- / Y-Dir-
      ANDD=   D300 D8340  ; X_Pick / X_Current
      ANDD=   D214 D8350  ; Z-Waiting / Z_Current
      ANDD=   K0 D8360  ; Y_Current
      MOV     K2 D620
92    LD      EnableInput
      AND     M622  ; Step2
      DDRVA   K-4800 D208 Y002 Y005
      ANDP    M8029
      MOV     K3 D620
118   LD      EnableInput
      AND     M623  ; Step3
      DDRVI   K14000 D206 Y001 Y004  ; F-Z LOAD
      ANDP    M8029
      MOV     K4 D620
144   LD      EnableInput
      AND     M624  ; Step4
      DDRVA   K0 D210 Y002 Y005  ; F-Y LOAD
      ANDP    M8029
      MOV     K5 D620
      OUT     Out1
171   LD      EnableInput
      AND     M625  ; Step5
      DDRVA   D224 D202 Y000 Y003  ; X_Fail / F-X LOAD
      DDRVA   D226 D206 Y001 Y004  ; Z_Fail
      ANDD=   D224 D8340  ; X_Fail / X_Current
      ANDD=   D226 D8350  ; Z_Fail / Z_Current
      MOV     K6 D620
230   LD      EnableInput
      AND     M626  ; Step6
      DDRVA   D228 D210 Y002 Y005  ; Y_Fail
      ANDP    M8029
      MOV     K7 D620
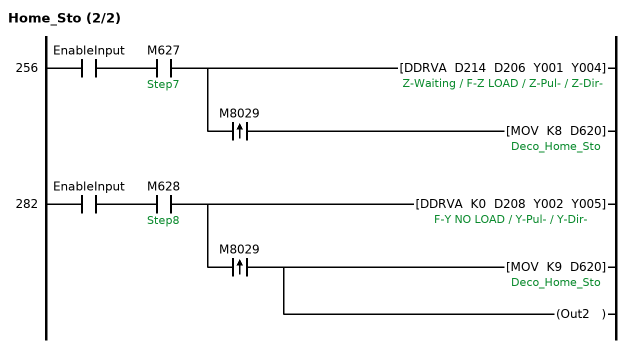
256   LD      EnableInput
      AND     M627  ; Step7
      DDRVA   D214 D206 Y001 Y004
      ANDP    M8029
      MOV     K8 D620
282   LD      EnableInput
      AND     M628  ; Step8
      DDRVA   K0 D208 Y002 Y005
      ANDP    M8029
      MOV     K9 D620
      OUT     Out2
END_FUNCTION_BLOCK

FUNCTION_BLOCK GoToFailPos
VAR_INPUT
  Enable_Input : BOOL;
END_VAR
VAR_OUTPUT
  Out1 : BOOL;
END_VAR
